// TIA Portal V19 export
TYPE "LAF_typeDevDiagModStateMode"
TITLE = PN device diag modul state / PN Device Diag Modul Status
// This data type contains the structure of the parameters and the return values of the moduls. / Struktur Modul Status
// stored: Access Published
   STRUCT
      laddr { ExternalAccessible := 'False'; ExternalVisible := 'False'; ExternalWritable := 'False'} : HW_DEVICE;   // Lokale Adresse / Local address
      mode { ExternalAccessible := 'False'; ExternalVisible := 'False'; ExternalWritable := 'False'} : UInt;   // Mode 1..5
      retVal { ExternalAccessible := 'False'; ExternalVisible := 'False'; ExternalWritable := 'False'} : Int;   // Rückmeldung / Return value
      state { ExternalAccessible := 'False'; ExternalVisible := 'False'; ExternalWritable := 'False'} : Array[0..127] of Bool;   // Array für bis 127 Module / Array for up to 127 modules
   END_STRUCT;
END_TYPE
